FUNCTION_BLOCK GreenMasterBase
VAR PERSISTENT
	Parameters: GreenMasterBaseParameters;
	ParametersSC: SmokeControlParametersBase;
	Simulation: Simulation;
END_VAR
VAR_INPUT
	EN: BOOL := TRUE;
	RemoteEN: BOOL;
	DI: GreenMasterDI_Base;
	AI: GreenMasterAI_Base;
	AI2: GreenMasterAIU_Base;
	TCP_AI: GreenMasterSmokeControl_Base;
	Reverse_C_QN1: BOOL := TRUE;
	NightCooling: BOOL;
	EnableFansAndDampers: BOOL := TRUE;
END_VAR
VAR_OUTPUT
	ENO: BOOL;
	VentilationRunning: BOOL;
	TemperatureControlRunning: BOOL;
END_VAR
VAR
	StateStartTime: LTIME;
	Ventilation: BOOL;
	SystemStateVentilation: BOOL;
	AlarmMonitor: AlarmMonitor;
	Hysteresis_0: Hysteresis;
	Hysteresis_1: Hysteresis;
	
	OvrTemperatureControl: BOOL;
	OvrTemperatureCV: REAL;
	Scale1: Scale;
	Scale2: Scale;
	Scale3: Scale;
	TemperatureController: PidController;
	TP1: TP;
	TON1: TON;
	C_QN1_Low: LREAL;
	C_QN1_High: LREAL;
	
	test: BOOL;
	Av: Average;
	Pump1_TON: TON;
	Pump2_TON: TON;
	FreezeControl: BOOL;
	FreezeControlENO: BOOL;
	TempCV: LREAL;
	FreezeControlCV: LREAL;
	FreezeController: PidController;
	Hysteresis_2: Hysteresis;
	Hysteresis_3: Hysteresis;
	Hysteresis_4: Hysteresis;
	FireAlarmExtractAirTemperatureHysteresis: Hysteresis;
	FireAlarmExtractAirPressureTemperatureHysteresis: Hysteresis;
	FireAlarmExtractAirPressureHysteresis: Hysteresis;
	WriteLRealOnlyIf_0: WriteLRealOnlyIf;
	ColdRecyclingHysteresis: Hysteresis;
	TempDevMon: DeviationMonitor;
	SupplyDevMon: DeviationMonitor;
	ExtractDevMon: DeviationMonitor;
END_VAR
VAR // added by the converter: edge detectors and wires of the graphical bodies
    _w1, _w2, _w4, _w5, _w6, _w7, _w8 : ANY;
    _w3 : BOOL;
END_VAR


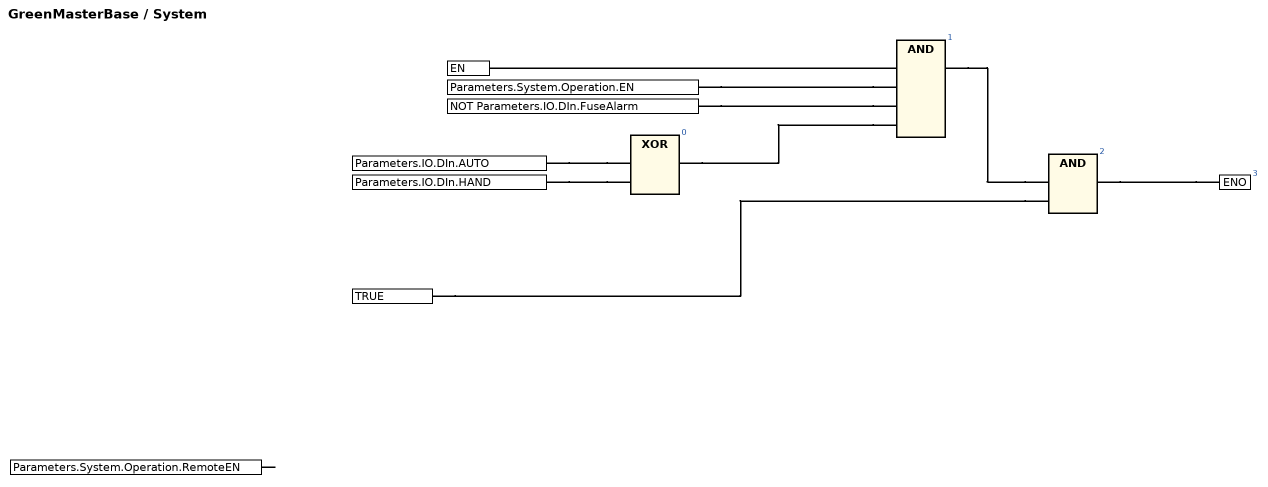
// PAGE System
ENO := (EN AND Parameters.System.Operation.EN AND (NOT Parameters.IO.DIn.FuseAlarm) AND (Parameters.IO.DIn.AUTO XOR Parameters.IO.DIn.HAND)) AND TRUE;

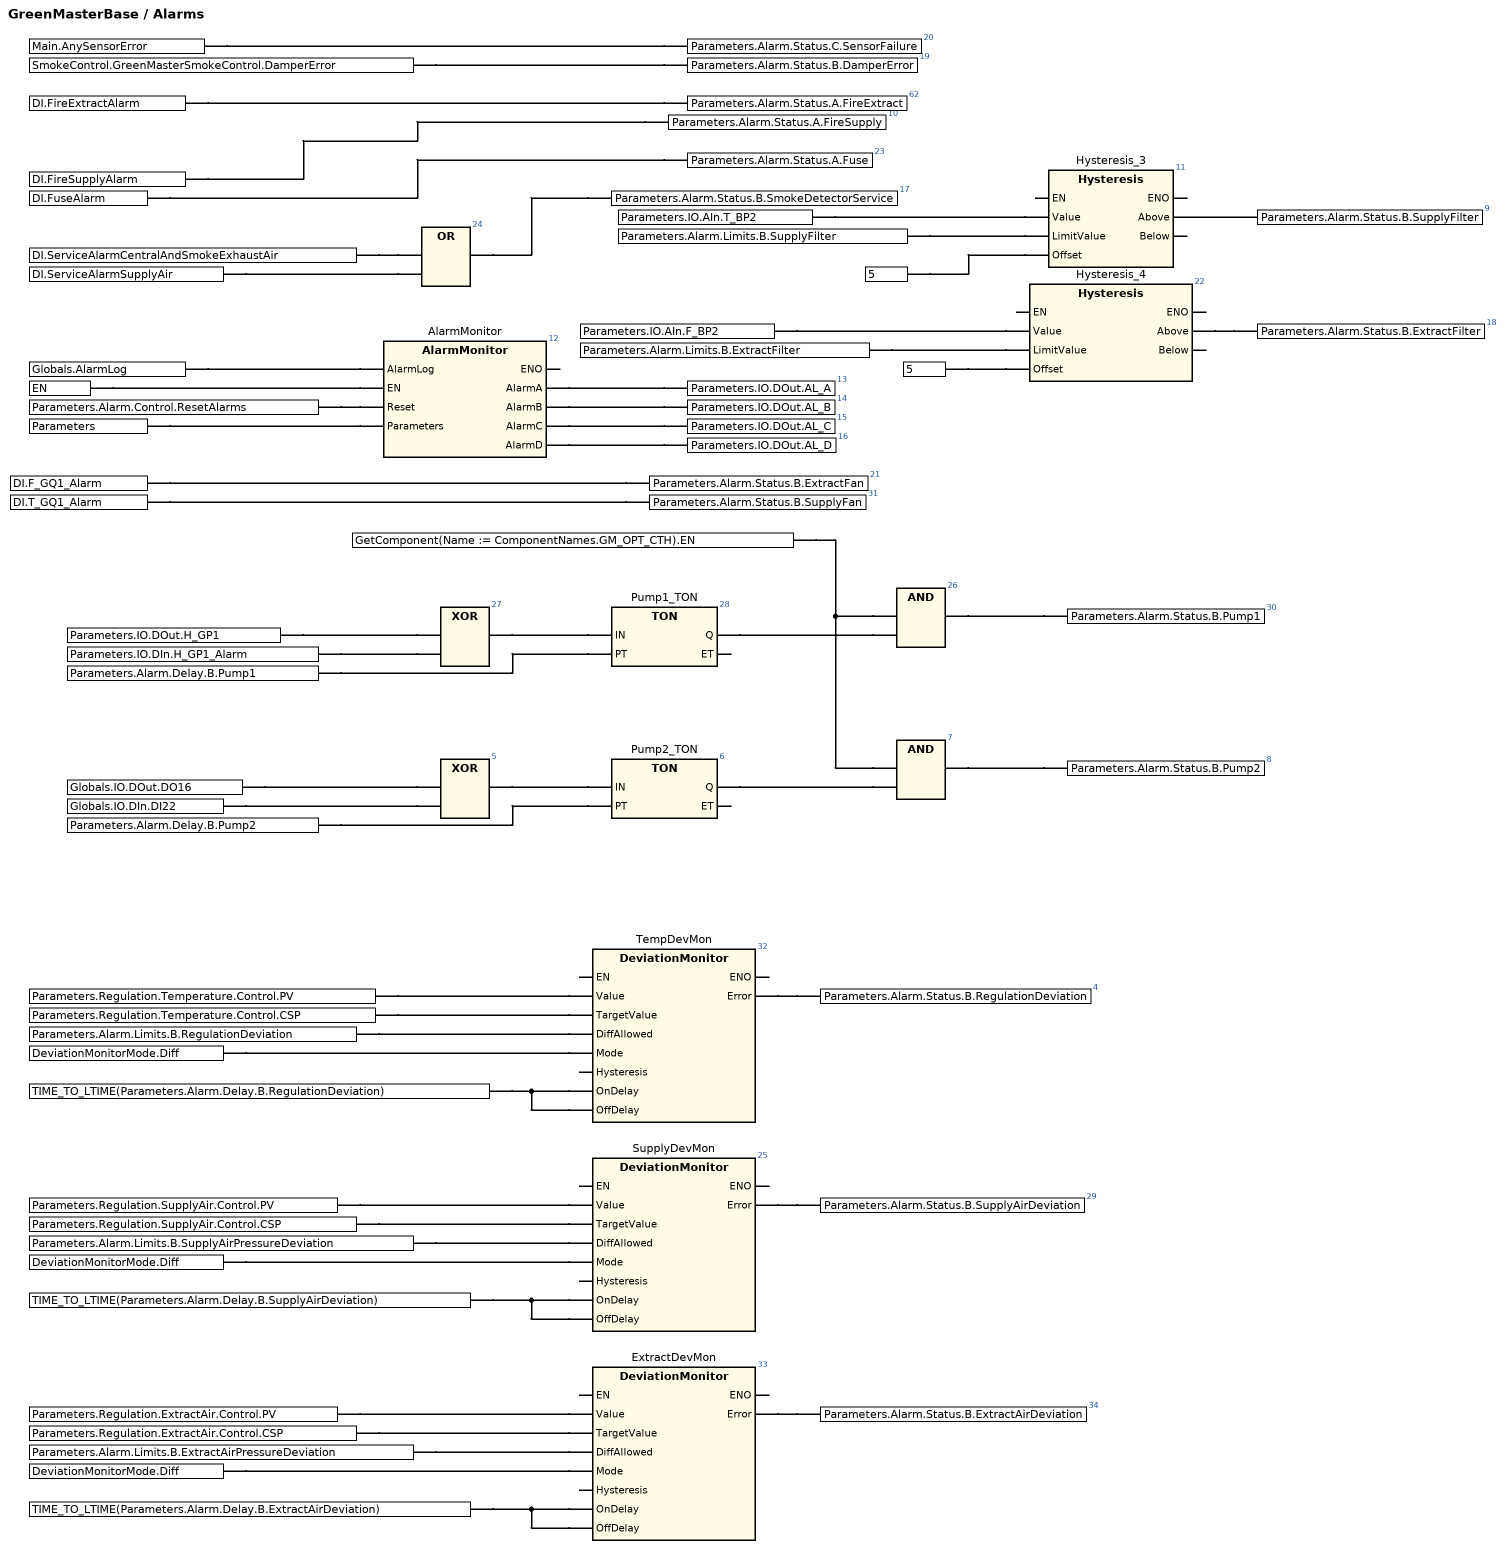
// PAGE Alarms
Parameters.Alarm.Status.B.RegulationDeviation := TempDevMon.Error;
Pump2_TON(IN := Globals.IO.DOut.DO16 XOR Globals.IO.DIn.DI22, PT := Parameters.Alarm.Delay.B.Pump2); // TON
Parameters.Alarm.Status.B.Pump2 := (GetComponent(Name := ComponentNames.GM_OPT_CTH).EN) AND Pump2_TON.Q;
Parameters.Alarm.Status.B.SupplyFilter := Hysteresis_3.Above;
Parameters.Alarm.Status.A.FireSupply := DI.FireSupplyAlarm;
Hysteresis_3(
    Value := Parameters.IO.AIn.T_BP2,
    LimitValue := Parameters.Alarm.Limits.B.SupplyFilter,
    Offset := 5); // Hysteresis
AlarmMonitor(
    AlarmLog := Globals.AlarmLog,
    EN := EN,
    Reset := Parameters.Alarm.Control.ResetAlarms,
    Parameters := Parameters);
Parameters.IO.DOut.AL_A := AlarmMonitor.AlarmA;
Parameters.IO.DOut.AL_B := AlarmMonitor.AlarmB;
Parameters.IO.DOut.AL_C := AlarmMonitor.AlarmC;
Parameters.IO.DOut.AL_D := AlarmMonitor.AlarmD;
Parameters.Alarm.Status.B.SmokeDetectorService := _w1;
Parameters.Alarm.Status.B.ExtractFilter := Hysteresis_4.Above;
Parameters.Alarm.Status.B.DamperError := SmokeControl.GreenMasterSmokeControl.DamperError;
Parameters.Alarm.Status.C.SensorFailure := Main.AnySensorError;
Parameters.Alarm.Status.B.ExtractFan := DI.F_GQ1_Alarm;
Hysteresis_4(
    Value := Parameters.IO.AIn.F_BP2,
    LimitValue := Parameters.Alarm.Limits.B.ExtractFilter,
    Offset := 5); // Hysteresis
Parameters.Alarm.Status.A.Fuse := DI.FuseAlarm;
_w1 := DI.ServiceAlarmCentralAndSmokeExhaustAir OR DI.ServiceAlarmSupplyAir;
SupplyDevMon(
    Value := Parameters.Regulation.SupplyAir.Control.PV,
    TargetValue := Parameters.Regulation.SupplyAir.Control.CSP,
    DiffAllowed := Parameters.Alarm.Limits.B.SupplyAirPressureDeviation,
    Mode := DeviationMonitorMode.Diff,
    OnDelay := TIME_TO_LTIME(Parameters.Alarm.Delay.B.SupplyAirDeviation),
    OffDelay := TIME_TO_LTIME(Parameters.Alarm.Delay.B.SupplyAirDeviation)); // DeviationMonitor
_w2 := (GetComponent(Name := ComponentNames.GM_OPT_CTH).EN) AND Pump1_TON.Q;
Pump1_TON(IN := Parameters.IO.DOut.H_GP1 XOR Parameters.IO.DIn.H_GP1_Alarm, PT := Parameters.Alarm.Delay.B.Pump1); // TON
Parameters.Alarm.Status.B.SupplyAirDeviation := SupplyDevMon.Error;
Parameters.Alarm.Status.B.Pump1 := _w2;
Parameters.Alarm.Status.B.SupplyFan := DI.T_GQ1_Alarm;
TempDevMon(
    Value := Parameters.Regulation.Temperature.Control.PV,
    TargetValue := Parameters.Regulation.Temperature.Control.CSP,
    DiffAllowed := Parameters.Alarm.Limits.B.RegulationDeviation,
    Mode := DeviationMonitorMode.Diff,
    OnDelay := TIME_TO_LTIME(Parameters.Alarm.Delay.B.RegulationDeviation),
    OffDelay := TIME_TO_LTIME(Parameters.Alarm.Delay.B.RegulationDeviation)); // DeviationMonitor
ExtractDevMon(
    Value := Parameters.Regulation.ExtractAir.Control.PV,
    TargetValue := Parameters.Regulation.ExtractAir.Control.CSP,
    DiffAllowed := Parameters.Alarm.Limits.B.ExtractAirPressureDeviation,
    Mode := DeviationMonitorMode.Diff,
    OnDelay := TIME_TO_LTIME(Parameters.Alarm.Delay.B.ExtractAirDeviation),
    OffDelay := TIME_TO_LTIME(Parameters.Alarm.Delay.B.ExtractAirDeviation)); // DeviationMonitor
Parameters.Alarm.Status.B.ExtractAirDeviation := ExtractDevMon.Error;

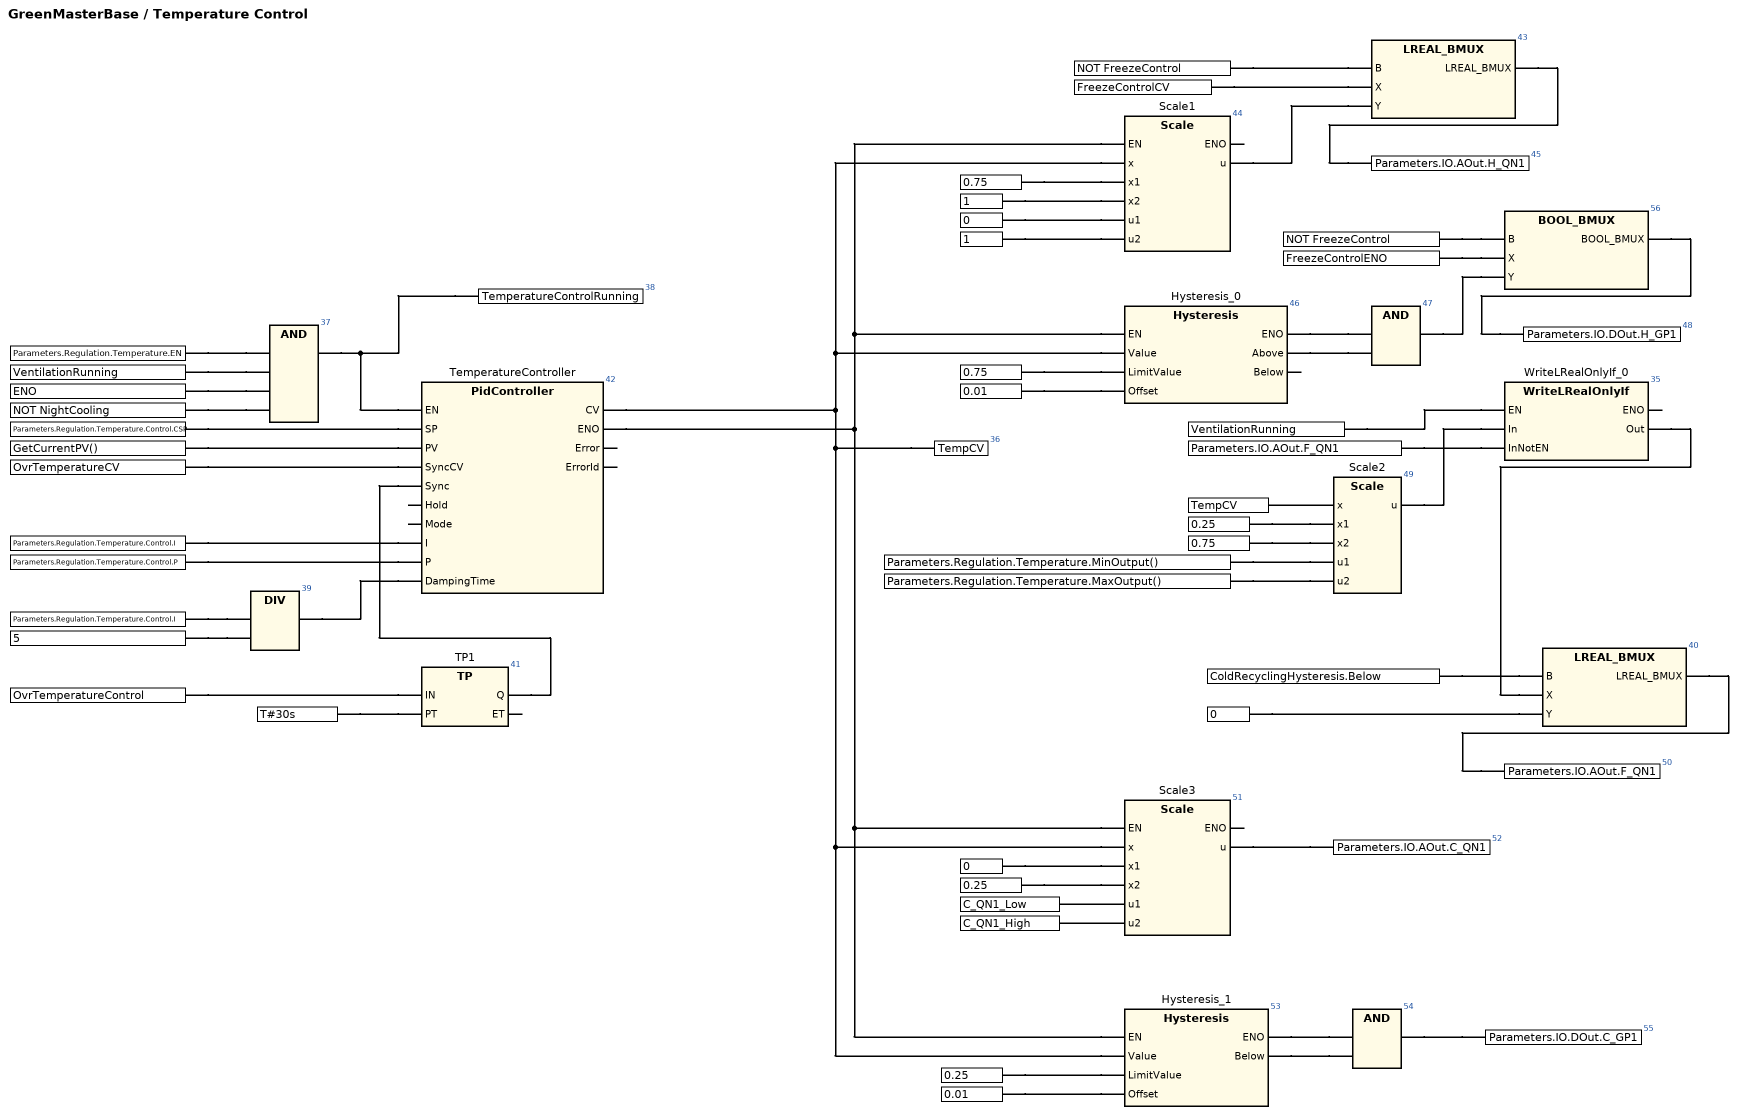
// PAGE Temperature Control
WriteLRealOnlyIf_0(EN := VentilationRunning, In := Scale2.u, InNotEN := Parameters.IO.AOut.F_QN1); // WriteLRealOnlyIf
TempCV := TemperatureController.CV;
_w3 := Parameters.Regulation.Temperature.EN AND VentilationRunning AND ENO AND (NOT NightCooling);
TemperatureControlRunning := _w3;
_w4 := Parameters.Regulation.Temperature.Control.I / 5;
_w5 := LREAL_BMUX(B := ColdRecyclingHysteresis.Below, X := WriteLRealOnlyIf_0.Out, Y := 0);
TP1(IN := OvrTemperatureControl, PT := T#30s); // TP
TemperatureController(
    EN := _w3,
    SP := Parameters.Regulation.Temperature.Control.CSP,
    PV := GetCurrentPV(),
    SyncCV := OvrTemperatureCV,
    Sync := TP1.Q,
    I := Parameters.Regulation.Temperature.Control.I,
    P := Parameters.Regulation.Temperature.Control.P,
    DampingTime := _w4); // PidController
_w6 := LREAL_BMUX(B := NOT FreezeControl, X := FreezeControlCV, Y := Scale1.u);
Scale1(EN := TemperatureController.ENO, x := TemperatureController.CV, x1 := 0.75, x2 := 1, u1 := 0, u2 := 1); // Scale
Parameters.IO.AOut.H_QN1 := _w6;
Hysteresis_0(
    EN := TemperatureController.ENO,
    Value := TemperatureController.CV,
    LimitValue := 0.75,
    Offset := 0.01); // Hysteresis
_w7 := Hysteresis_0.ENO AND Hysteresis_0.Above;
Parameters.IO.DOut.H_GP1 := _w8;
Scale2(
    x := TempCV,
    x1 := 0.25,
    x2 := 0.75,
    u1 := Parameters.Regulation.Temperature.MinOutput(),
    u2 := Parameters.Regulation.Temperature.MaxOutput()); // Scale
Parameters.IO.AOut.F_QN1 := _w5;
Scale3(
    EN := TemperatureController.ENO,
    x := TemperatureController.CV,
    x1 := 0,
    x2 := 0.25,
    u1 := C_QN1_Low,
    u2 := C_QN1_High); // Scale
Parameters.IO.AOut.C_QN1 := Scale3.u;
Hysteresis_1(
    EN := TemperatureController.ENO,
    Value := TemperatureController.CV,
    LimitValue := 0.25,
    Offset := 0.01); // Hysteresis
Parameters.IO.DOut.C_GP1 := Hysteresis_1.ENO AND Hysteresis_1.Below;
_w8 := BOOL_BMUX(B := NOT FreezeControl, X := FreezeControlENO, Y := _w7);

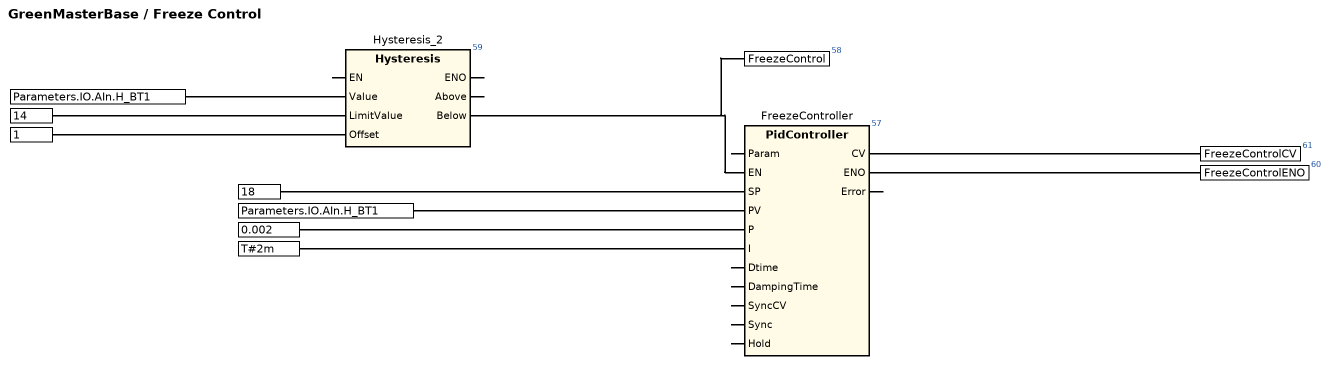
// PAGE Freeze Control
FreezeController(EN := Hysteresis_2.Below, SP := 18, PV := Parameters.IO.AIn.H_BT1, P := 0.002, I := T#2m); // PidController
FreezeControl := Hysteresis_2.Below;
Hysteresis_2(Value := Parameters.IO.AIn.H_BT1, LimitValue := 14, Offset := 1); // Hysteresis
FreezeControlENO := FreezeController.ENO;
FreezeControlCV := FreezeController.CV;

// PAGE Alarms
Parameters.Alarm.Status.A.FireExtract := DI.FireExtractAlarm;
// Parameters.System.Operation.RemoteEN: input not connected

METHOD CloseDampers : BOOL
VAR_INPUT
END_VAR
Parameters.IO.DOut.T_QM2 := FALSE;
Parameters.IO.DOut.F_QM1 := FALSE;
Parameters.IO.DOut.F_QM2 := TRUE;
Parameters.IO.DOut.R_QM1 := FALSE;
Parameters.IO.DOut.T_QM1_1 := FALSE;
Parameters.IO.DOut.T_QM1_2 := FALSE;
Parameters.IO.DOut.T_QM1_3 := FALSE;
Parameters.IO.DOut.T_QM1_4 := FALSE;
Parameters.IO.DOut.T_QM1_5 := FALSE;
Parameters.IO.DOut.T_QM1_6 := FALSE;
END_METHOD

METHOD DampersOpen : BOOL
VAR_INPUT
END_VAR
DampersOpen := Parameters.IO.DOut.T_QM2_OnTime > LTIME#30s and Parameters.IO.DOut.F_QM1_OnTime > LTIME#30s;
END_METHOD

METHOD ExtractFanOverride : BOOL
VAR_INPUT
	Override: BOOL;
	Speed: LREAL;
END_VAR
END_METHOD

METHOD FB_init : BOOL
VAR_INPUT
	bInitRetains : BOOL; // if TRUE, the retain variables are initialized (warm start / cold start)
	bInCopyCode : BOOL;  // if TRUE, the instance afterwards gets moved into the copy code (online change)
END_VAR
IF bInitRetains THEN
	Parameters.Regulation.Temperature.Control.SP := 20;	
	Parameters.Regulation.SupplyAir.Control.SP := 100;	
	Parameters.Regulation.ExtractAir.Control.SP := 100;	
	Parameters.Regulation.SupplyAir.Control.SP_HighSpeed := 100;	
	Parameters.Regulation.ExtractAir.Control.SP_HighSpeed := 100;	
END_IF
END_METHOD

METHOD Fire : BOOL
VAR_INPUT
END_VAR
Parameters.IO.DOut.F_QM2 := FALSE;
Fire := TRUE;
END_METHOD

METHOD FireAlarm : BOOL
VAR_INPUT
END_VAR
VAR_INST
END_VAR
FireAlarm := Parameters.Alarm.Active.A.FireExtract OR 
	Parameters.Alarm.Active.A.FireSupply OR
	Parameters.Alarm.Active.A.FireExtractPressure OR
	Parameters.Alarm.Active.A.FireExtractTemperature OR
	Parameters.Alarm.Active.A.FireExtractExternal;
END_METHOD

METHOD FireEnd : BOOL
VAR_INPUT
END_VAR
Parameters.IO.DOut.F_QM2 := TRUE;
END_METHOD

METHOD FireSupply : BOOL
VAR_INPUT
END_VAR
FireSupply := TRUE;
END_METHOD

METHOD FireSupplyEnd : BOOL
VAR_INPUT
END_VAR
END_METHOD

{attribute 'TcEncoding':='UTF-8'}
METHOD GetActiveStateName : string
VAR_INPUT
END_VAR
GetActiveStateName := '';
END_METHOD

METHOD GetCurrentExtractAirPV : LREAL
VAR_INPUT
END_VAR

IF Parameters.Regulation.ExtractAir.ControlMode =  FanControlTypes.Pressure  THEN
	GetCurrentExtractAirPV := AI2.F_BP1;
ELSE
	GetCurrentExtractAirPV := AI2.F_BF1;
END_IF
END_METHOD

METHOD GetCurrentExtractAirSP : LREAL
VAR_INPUT
END_VAR
CASE Parameters.System.Operation.Mode OF
	SystemStatesRunMode.Off:
		GetCurrentExtractAirSP := 0;

	SystemStatesRunMode.LowSpeed:
		GetCurrentExtractAirSP := Parameters.Regulation.ExtractAir.Control.SP + Parameters.Regulation.ExtractAir.SetPointAdjustment.Y;

	SystemStatesRunMode.HighSpeed:
		GetCurrentExtractAirSP := Parameters.Regulation.ExtractAir.Control.SP_HighSpeed + Parameters.Regulation.ExtractAir.SetPointAdjustment.Y;

END_CASE
END_METHOD

METHOD GetCurrentPV : LREAL
VAR_INPUT
END_VAR
GetCurrentPV := AI.T_BT1;
IF Parameters.Regulation.Temperature.TemperatureControlSource = TemperatureControlSources.F_BT1 THEN
	GetCurrentPV := AI.F_BT1;
ELSIF Parameters.Regulation.Temperature.TemperatureControlSource = TemperatureControlSources.BT2 THEN
	GetCurrentPV := AI.BT2;
END_IF
END_METHOD

METHOD GetCurrentSP : LREAL
VAR_INPUT
END_VAR
IF Parameters.Regulation.Temperature.TemperatureControlSource = TemperatureControlSources.F_BT1 THEN
	GetCurrentSP := Parameters.Regulation.Temperature.Control.SP + Parameters.Regulation.Temperature.SetPointAdjustment.Y;
ELSE
	GetCurrentSP := Parameters.Regulation.Temperature.Control.SP;
END_IF
END_METHOD

METHOD GetCurrentSupplyAirPV : LREAL
VAR_INPUT
END_VAR

IF Parameters.Regulation.SupplyAir.ControlMode =  FanControlTypes.Pressure  THEN
	GetCurrentSupplyAirPV := AI2.T_BP1;
ELSE
	GetCurrentSupplyAirPV := AI2.T_BF1;
END_IF
END_METHOD

METHOD GetCurrentSupplyAirSP : LREAL
VAR_INPUT
END_VAR
END_METHOD

METHOD GetFireExtractAlarms : BOOL
VAR_INPUT
END_VAR
GetFireExtractAlarms := Parameters.Alarm.Active.A.FireExtract OR
	Parameters.Alarm.Active.A.FireExtractPressure OR
	Parameters.Alarm.Active.A.FireExtractTemperature OR
	Parameters.Alarm.Active.A.FireExtractExternal;
END_METHOD

METHOD GetParameters : reference to GreenMasterBaseParameters
VAR_INPUT
END_VAR
GetParameters REF= Parameters;
END_METHOD

METHOD GetParametersSC : reference to SmokeControlParametersBase
VAR_INPUT
END_VAR
GetParametersSC REF= ParametersSC;
END_METHOD

METHOD Runnable : BOOL
VAR_INPUT
END_VAR
Runnable := ENO and not (Parameters.Alarm.Active.B.ExtractFan or Parameters.Alarm.Active.B.SupplyFan);
END_METHOD

METHOD Simulate : BOOL
VAR_INPUT
	Parameters: reference to GreenMasterBaseParameters;
END_VAR

VAR
	
END_VAR

VAR_INST
	FirstTime: BOOL;
END_VAR
IF NOT FirstTime THEN
	Parameters.IO.DIn.FireSupplyAlarm := TRUE;
	Parameters.IO.DIn.FuseAlarm := TRUE;
	FirstTime := TRUE;
END_IF

Parameters.IO.DIn.F_QM2_Closed := Parameters.IO.DOut.F_QM2_OnTime < LTIME#5S; 
Parameters.IO.DIn.F_QM2_Open := Parameters.IO.DOut.F_QM2_OnTime > LTIME#30S;
END_METHOD

METHOD StateTime : LTIME
VAR_INPUT
END_VAR
StateTime := LTIME() - StateStartTime;
END_METHOD

METHOD SupplyFanOverride : BOOL
VAR_INPUT
	Override: BOOL;
	Speed: LREAL;
END_VAR
END_METHOD

METHOD SystemStateST : BOOL
VAR_IN_OUT
	Parameters: GreenMasterBaseParameters;
END_VAR
VAR_INPUT
END_VAR
VAR_INST
	SystemStateSTInitDone: BOOL;
	CurrentStateTime: LTIME;
END_VAR
VAR_INST
	State: REFERENCE TO SystemStates;
	NextState: SystemStates;	
END_VAR
VAR
	LogStr: string;
END_VAR
State REF= Parameters.System.Operation.State;
IF NOT SystemStateSTInitDone THEN
	SystemStateStarted();
	State := SystemStates.Idle;	
	SystemStateSTInitDone := TRUE;
END_IF

IF NextState <> State THEN
	LogStr := 'Entering state ';
	LogStr := Concat(LogStr, TO_STRING(NextState));
	Main.EventLog.LogEvent(Message := LogStr, Kind := EventTypes.Information);
	SystemStateStarted();
	// Entry state logic
	CASE NextState OF

		SystemStates.Start:
			;
			
		SystemStates.Idle:
			SystemStateVentilation := FALSE;
			Parameters.IO.DOut.F_QM1 := FALSE;
			Parameters.IO.DOut.T_QM2 := FALSE;
			Parameters.IO.AOut.F_QN1 := 0;
			Parameters.IO.AOut.F_GQ1 := 0;
			Parameters.IO.AOut.T_GQ1 := 0;
			Parameters.IO.DOut.T_QM1_1 := FALSE;
			Parameters.IO.DOut.T_QM1_2 := FALSE;
			Parameters.IO.DOut.T_QM1_3 := FALSE;
			Parameters.IO.DOut.T_QM1_4 := FALSE;
			Parameters.IO.DOut.T_QM1_5 := FALSE;
			Parameters.IO.DOut.T_QM1_6 := FALSE;
			Parameters.IO.AOut.F_GQ1 := 0;
			Parameters.IO.AOut.T_GQ1 := 0;
			ExtractFanOverride(FALSE, 0);
			SupplyFanOverride(FALSE, 0);
			
		SystemStates.OpenDampers:
			Parameters.IO.AOut.F_QN1 := 0;

		SystemStates.StartupHeatRecovery:
			OvrTemperatureCV := 0.5;
			
		SystemStates.Run:
			SystemStateVentilation := TRUE;

		SystemStates.FireHandling:
			;

		SystemStates.FireExhaust:
			Parameters.IO.DOut.F_QM1 := FALSE;
			Parameters.IO.DOut.F_QM2 := FALSE;
			Parameters.IO.DOut.T_QM2 := TRUE;
			Parameters.IO.DOut.T_QM1_1 := TRUE;
			Parameters.IO.DOut.T_QM1_2 := TRUE;
			Parameters.IO.DOut.T_QM1_3 := TRUE;
			Parameters.IO.DOut.T_QM1_4 := TRUE;
			Parameters.IO.DOut.T_QM1_5 := TRUE;
			Parameters.IO.DOut.T_QM1_6 := TRUE;
			Fire();
				
		SystemStates.FireSupply:
			FireSupply();	
			Parameters.IO.DOut.F_QM1 := FALSE;
			Parameters.IO.DOut.F_QM2 := TRUE;
			Parameters.IO.DOut.T_QM2 := FALSE;
			Parameters.IO.DOut.T_QM1_1 := FALSE;
			Parameters.IO.DOut.T_QM1_2 := FALSE;
			Parameters.IO.DOut.T_QM1_3 := FALSE;
			Parameters.IO.DOut.T_QM1_4 := FALSE;
			Parameters.IO.DOut.T_QM1_5 := FALSE;
			Parameters.IO.DOut.T_QM1_6 := FALSE;

		SystemStates.Ventilate:
			;

		SystemStates.Exercise:
			SystemStateVentilation := FALSE;
	END_CASE;
end_if;

State := NextState;
CurrentStateTime := StateTime();

// Do while in state logic
CASE State OF

	SystemStates.Start:
		;
		
	SystemStates.Idle:
		Parameters.System.Operation.Mode := SystemStatesRunMode.Off;
		IF StateTime() > LTIME#30S THEN
			CloseDampers();
		END_IF
		
	SystemStates.OpenDampers:
		Parameters.IO.DOut.F_QM1 := TRUE;		
		Parameters.IO.DOut.F_QM2 := TRUE;
		Parameters.IO.DOut.R_QM1 := FALSE;
		;

	SystemStates.StartupHeatRecovery:
		IF StateTime() > Parameters.System.Operation.ExhaustFanStartupDelay THEN
			ExtractFanOverride(TRUE, Parameters.Regulation.ExtractAir.StartupFanSpeed);
			//Parameters.IO.AOut.F_GQ1 := Parameters.Regulation.ExtractAir.StartupFanSpeed;			
			Parameters.IO.DOut.T_QM2 := TRUE;
			Parameters.IO.DOut.T_QM1_1 := TRUE;
			Parameters.IO.DOut.T_QM1_2 := TRUE;
			Parameters.IO.DOut.T_QM1_3 := TRUE;
			Parameters.IO.DOut.T_QM1_4 := TRUE;
			Parameters.IO.DOut.T_QM1_5 := TRUE;
			Parameters.IO.DOut.T_QM1_6 := TRUE;
		END_IF
		IF StateTime() > Parameters.System.Operation.SupplyFanStartupDelay THEN
			SupplyFanOverride(TRUE, Parameters.Regulation.ExtractAir.StartupFanSpeed);
			//Parameters.IO.AOut.T_GQ1 := Parameters.Regulation.SupplyAir.StartupFanSpeed;			
		END_IF
		OvrTemperatureControl := (StateTime() > LTIME#1000MS) AND (StateTime() < LTIME#2000MS);
		
	SystemStates.Run:
		
		ExtractFanOverride(FALSE, 0);
		SupplyFanOverride(FALSE, 0);
		Parameters.System.Operation.Mode := SystemStatesRunMode.LowSpeed;
		IF Parameters.Regulation.Temperature.ColdRecycling.EN THEN
			ColdRecyclingHysteresis(Value := Parameters.IO.AIn.F_BT1, LimitValue := Parameters.Regulation.CompensationTemperature + Parameters.Regulation.Temperature.ColdRecycling.Offset, Offset := Parameters.Regulation.Temperature.ColdRecycling.Hysteresis);
			IF ColdRecyclingHysteresis.Below THEN
				Parameters.IO.AOut.F_QN1 := 0;	
			ELSE				
				Parameters.IO.AOut.F_QN1 := 1;	
			END_IF
		END_IF

	SystemStates.FireHandling:
		;

	SystemStates.FireExhaust:
		ADS_Standard.Tags.Settings.T_GQ1_M := FALSE;
		ADS_Standard.Tags.Settings.F_GQ1_M := FALSE;
		ADS_Standard.Tags.Settings.H_QN1_M := FALSE;
		ADS_Standard.Tags.Settings.TX1_M := FALSE;
		ADS_Standard.Tags.Settings.C_QN1_M := FALSE;
			
	SystemStates.FireSupply:
		ADS_Standard.Tags.Settings.T_GQ1_M := FALSE;
		ADS_Standard.Tags.Settings.F_GQ1_M := FALSE;
		ADS_Standard.Tags.Settings.H_QN1_M := FALSE;
		ADS_Standard.Tags.Settings.TX1_M := FALSE;
		ADS_Standard.Tags.Settings.C_QN1_M := FALSE;

	SystemStates.Ventilate:
		;

	SystemStates.Exercise:
		;
end_case;

// Transitions

IF (State <> SystemStates.FirePanel) AND Main.CTH_Interface.FirePanelActive AND Main.CTH_Interface.EN THEN
	NextState := SystemStates.FirePanel;		
END_IF

CASE State OF

	SystemStates.None:
		NextState := SystemStates.Start;
 
	SystemStates.Start:
		NextState := SystemStates.Idle;
		
	SystemStates.Idle:
		if FireAlarm() then
			NextState := SystemStates.FireHandling;
		end_if;
		IF Runnable() THEN
			NextState := SystemStates.OpenDampers;
		end_if;
		
	SystemStates.OpenDampers:
		if FireAlarm() then
			NextState := SystemStates.FireHandling;
		end_if;
		IF StateTime() > LTIME#30S THEN
			NextState := SystemStates.StartupHeatRecovery;
		end_if;
		IF NOT Runnable() THEN
			NextState := SystemStates.Idle;
		end_if;

	SystemStates.StartupHeatRecovery:
		if FireAlarm() then
			NextState := SystemStates.FireHandling;
		end_if;
		IF NOT Runnable() THEN
			NextState := SystemStates.Idle;
		END_IF;
		IF StateTime() > Parameters.System.Operation.StartupHeatRecoveryTime THEN
			NextState := SystemStates.Run;
		END_IF;
		
	SystemStates.Run:
		if FireAlarm() then
			NextState := SystemStates.FireHandling;
		end_if;
			
		IF NOT Runnable() THEN
			NextState := SystemStates.PostRun;
		end_if;
		IF SmokeControl.Exercising THEN
			NextState := SystemStates.Exercise;
		end_if;

	SystemStates.PostRun:
		if FireAlarm() then
			NextState := SystemStates.FireHandling;
		end_if;
		IF NOT Runnable() THEN
			NextState := SystemStates.Idle;
		end_if;
		IF StateTime() > Parameters.System.Operation.PostVentilationTime THEN
			NextState := SystemStates.Idle;
		end_if;
		
	SystemStates.FireHandling:
		FireAlarm();
		IF Parameters.Alarm.Active.A.FireSupply AND NOT GetFireExtractAlarms() THEN
			NextState := SystemStates.FireSupply;
		ELSIF GetFireExtractAlarms() THEN
			NextState := SystemStates.FireExhaust;
		ELSE
			NextState := SystemStates.FireHandlingExit;			
		END_IF;
		
	SystemStates.FireHandlingExit:
		FireAlarm();
		NextState := SystemStates.Idle;

	SystemStates.FireExhaust:
		FireAlarm();
		IF NOT Parameters.Alarm.Active.A.FireSupply AND NOT GetFireExtractAlarms() THEN
			NextState := SystemStates.Ventilate;
		end_if;
		IF Parameters.Alarm.Active.A.FireSupply AND NOT GetFireExtractAlarms() THEN
			NextState := SystemStates.FireSupply;
		end_if;
			
	SystemStates.FireSupply:
		FireAlarm();
		IF GetFireExtractAlarms() THEN
			NextState := SystemStates.FireExhaust;
		end_if;
		IF NOT Parameters.Alarm.Active.A.FireSupply THEN
			NextState := SystemStates.FireHandlingExit;
		end_if;

	SystemStates.Ventilate:
		FireAlarm();
		IF NOT Parameters.Alarm.Active.A.FireSupply AND GetFireExtractAlarms() THEN
			NextState := SystemStates.FireExhaust;
		END_IF;
		IF Parameters.Alarm.Active.A.FireSupply THEN
			NextState := SystemStates.FireSupply;
		END_IF
		IF TRUE (* StateTime() > Parameters.System.Operation.PostFireVentilationTime *) THEN
			NextState := SystemStates.FireHandlingExit;
		END_IF;
		
	SystemStates.FirePanel:
		FireAlarm();
		IF NOT Main.CTH_Interface.FirePanelActive AND Main.CTH_Interface.EN  THEN
			NextState := SystemStates.Idle;		
		END_IF;
	
	SystemStates.Exercise:
		FireAlarm();
		IF NOT SmokeControl.Exercising  THEN
			NextState := SystemStates.Idle;		
		END_IF;
END_CASE;

IF NextState <> State THEN

	// Exit state logic
	CASE State OF

		SystemStates.Start:
			;
			
		SystemStates.Idle:
			;
			
		SystemStates.OpenDampers:
			;

		SystemStates.StartupHeatRecovery:
			OvrTemperatureControl := TRUE;	
			
		SystemStates.Run:
			;

		SystemStates.FireHandling:
			;

		SystemStates.FireExhaust:
			FireEnd();
				
		SystemStates.FireSupply:
			FireSupplyEnd();

		SystemStates.Ventilate:
			;

	end_case;
end_if;
END_METHOD

METHOD SystemStateStarted : BOOL
VAR_INPUT
END_VAR
StateStartTime := LTIME();
END_METHOD

METHOD Update : BOOL
VAR_INPUT
	DO_: REFERENCE TO GreenMasterDO_Base;
	AO: REFERENCE TO GreenMasterAO_Base;
END_VAR

VAR_INST
	FirstTime: BOOL;
END_VAR
IF NOT FirstTime THEN
	FirstTime := TRUE;
END_IF

FireAlarmExtractAirTemperatureHysteresis(Value := Parameters.IO.AIn.F_BT1,
	LimitValue := Parameters.Alarm.Limits.A.FireExtractTemperature,
	Offset := 1);
	
FireAlarmExtractAirPressureTemperatureHysteresis(Value := Parameters.IO.AIn.F_BT1,
	LimitValue := Parameters.Alarm.Limits.A.FireExtractPressureTemperature,
	Offset := 1);
	
FireAlarmExtractAirPressureHysteresis(Value := Parameters.IO.AIn.F_BP2,
	LimitValue := Parameters.Alarm.Limits.A.FireExtractPressure,
	Offset := 10);
	
Parameters.Alarm.Status.A.FireExtractTemperature := FireAlarmExtractAirTemperatureHysteresis.Above;
Parameters.Alarm.Status.A.FireExtractPressure := FireAlarmExtractAirPressureTemperatureHysteresis.Above AND
	FireAlarmExtractAirPressureHysteresis.Above;

IF Reverse_C_QN1 THEN
	C_QN1_Low := 1;
	C_QN1_High := 0;
ELSE
	C_QN1_Low := 0;
	C_QN1_High := 1;
END_IF

UpdateIO(DO_ := DO_, AO := AO);

IF Parameters.System.Operation.Simulation THEN
	Simulate(Parameters := Parameters);
END_IF

SystemStateST(Parameters := Parameters);

Parameters(GreenMaster := THIS^);
END_METHOD

METHOD UpdateIO : BOOL
VAR_INPUT
	DO_: REFERENCE TO GreenMasterDO_Base;
	AO: REFERENCE TO GreenMasterAO_Base;
END_VAR
Parameters.IO.AIn();
Parameters.IO.AOut();
Parameters.IO.DIn();
Parameters.IO.DOut();

Parameters.IO.AIn.Update(AI := AI, AI2 := AI2, Parameters := Parameters);
Parameters.IO.AOut.Update(AO := AO, Parameters := Parameters);
Parameters.IO.DIn.Update(DI := DI, Parameters := Parameters);
Parameters.IO.DOut.Update(DO_ := DO_, Parameters := Parameters, EnableWriteDampers := EnableFansAndDampers);
END_METHOD

END_FUNCTION_BLOCK

(* stored: Version 1.1.0.1, ProductVersion 3.1.4024.6
   POU GreenMasterBase: Id {3964931c-0c74-4f82-aa73-a9f5913e638a}, SpecialFunc None
   Method CloseDampers: Id {2b41e423-3c19-417f-b352-519030139e47}
   Method DampersOpen: Id {c8ec3299-3d43-469f-adbf-c5c4058ebc5b}
   Method ExtractFanOverride: Id {d4dae123-f430-4cea-bdb9-c30106c5f05d}
   Method FB_init: Id {1e201abe-9496-47c9-ad21-240006067df9}
   Method Fire: Id {bcae5a50-2529-4281-8457-a2544f030719}
   Method FireAlarm: Id {4d2863ab-7dbc-43e0-87de-bc6423403802}
   Method FireEnd: Id {1b0ca051-fe3f-4e93-97ea-c5e81688d583}
   Method FireSupply: Id {41b0c9c1-2722-44af-9ce2-69d4beaf887a}
   Method FireSupplyEnd: Id {f74128eb-b4b5-4e0e-9a00-0b445bdcc062}
   Method GetActiveStateName: Id {e67d6599-d64a-49bb-afd0-c8168047c7c8}
   Method GetCurrentExtractAirPV: Id {53abd77a-8c57-4316-ac40-e64f2159e488}
   Method GetCurrentExtractAirSP: Id {b10f141a-c01e-419f-90fd-692328c8afad}
   Method GetCurrentPV: Id {54dd4c5c-8873-45c5-8a20-5341e8f1cf37}
   Method GetCurrentSP: Id {9057130d-7737-4609-a28d-94fa4e95412d}
   Method GetCurrentSupplyAirPV: Id {70bc7f2a-64cc-4bba-b9d1-98ad82305898}
   Method GetCurrentSupplyAirSP: Id {e5d65448-6f20-4d77-b2e7-697b7a17cc5a}
   Method GetFireExtractAlarms: Id {c1708675-53aa-4624-a947-b3694b3cd0ec}
   Method GetParameters: Id {0b4dd537-bffd-4a45-a167-901028c44591}
   Method GetParametersSC: Id {3224ff51-720a-4182-90f0-3d33da53d667}
   Method Runnable: Id {60dd4a36-2d40-48ae-9dcb-3012f065c445}
   Method Simulate: Id {2c7e379c-c1c7-4206-9735-f2160708f434}
   Method StateTime: Id {16af60a9-8fdb-41dd-abaf-3111b1142416}
   Method SupplyFanOverride: Id {63286f14-74e9-40cd-8041-bfbc6adf3fb9}
   Method SystemStateST: Id {9bc36e52-b0aa-4d7d-90b3-a08e80d6b909}
   Method SystemStateStarted: Id {ba7965e0-3b5e-4542-8e64-3b6f30fe5aa6}
   Method Update: Id {329fda58-d838-4466-baad-8fd32e798b27}
   Method UpdateIO: Id {f79be100-de31-494f-aa80-cd5102c7087c} *)
